FUNCTION_BLOCK TankCtrl_Enabled EXTENDS _TankCtrl_State IMPLEMENTS I_Call

METHOD PRIVATE _GetTank : Result
VAR_INPUT
	iTag		: I_Tag;
END_VAR
VAR_OUTPUT
	iTank		: I_Domain;
END_VAR
VAR
	i			: GenIter(0);
END_VAR
_GetTank := GetDom(iTag, iDomain => iTank);
END_METHOD

METHOD Call
VAR_INPUT
	iTag	: Broadcast.Tags.I_Tag;
END_VAR
IF _ctx.priv.iTank <> 0 AND_THEN _ctx.priv.iTank.Tag = iTag THEN
	RETURN;
END_IF

IF NOT _ctx.priv.tankBuffer.Has(iTag) THEN
	_ctx.priv.tankBuffer.Push(iTag);
	_ctx.priv.sTankId := iTag.Option;
END_IF
END_METHOD

METHOD OnExecute
VAR
	iTag		: I_Tag;
	eResult		: Result;
END_VAR
IF _ctx.hmi.bMultiButton THEN
	_ctx.hmi.bMultiButton := FALSE;
	
	_ctx.priv.smgr.Request(_ctx.state.iDisabled);
	RETURN;
END_IF

IF IsOk(_ctx.priv.tankBuffer.Pop(iTag => iTag)) THEN
	IF IsOk(_GetTank(iTag, iTank => _ctx.priv.iTank), eCarry => eResult) THEN
		_ctx.priv.smgr.Request(_ctx.state.iFilling);
	ELSE
		CASE eResult OF
			None:
				// This can be used for log a failed request
			ELSE // Error
				// This can be used for log an incorrect argument
		END_CASE
	END_IF 
END_IF
END_METHOD

METHOD OnInit
_ctx.hmi.bMultiButtonVis := TRUE;
_ctx.hmi.nMultiButtonColor := COL.WHITE.Raw;
_ctx.hmi.nMultiButtonText := 'Press to Disable';

_ctx.priv.IsSystemOn.Rise();

_ctx.io.out.bRunPump := FALSE;

_ctx.priv.iTank := 0;
END_METHOD

END_FUNCTION_BLOCK

(* stored: Version 1.1.0.1
   POU TankCtrl_Enabled: Id {5cee1e32-2a64-48a5-b248-872a66806b16}, SpecialFunc None
   Method _GetTank: Id {b9443d87-d18f-45de-8de0-feecd1e722fa}
   Method Call: Id {15261221-0b6b-405c-ac53-e6f58082049a}
   Method OnExecute: Id {2c71692e-4c78-496f-9720-ad58d64c5078}
   Method OnInit: Id {18fecd57-2df1-483b-a2df-58a0e2543e29} *)
